(* PLC project Unnamed, Unknown Unnamed 1 *)
(* stored: creationDateTime 2024-01-09T16:45:07, modificationDateTime 2024-01-23T14:31:54 *)

FUNCTION_BLOCK Reals_Min
  VAR_INPUT
    u1 : REAL;
    u2 : REAL;
  END_VAR
  VAR_OUTPUT
    y : REAL;
  END_VAR

						y := min(u1, u2);
					
END_FUNCTION_BLOCK

FUNCTION_BLOCK Reals_MultiplyByParameter
  VAR_INPUT
    u : REAL;
    k : REAL;
  END_VAR
  VAR_OUTPUT
    y : REAL;
  END_VAR

						y := k * u;
					
END_FUNCTION_BLOCK

PROGRAM CustomPWithLimiter
  VAR_INPUT
    e : REAL;
    yMax : REAL;
  END_VAR
  VAR_OUTPUT
    y : REAL;
  END_VAR
  VAR
    gain : Reals_MultiplyByParameter;
    minValue : Reals_Min;
    k : REAL := 2.0;
  END_VAR

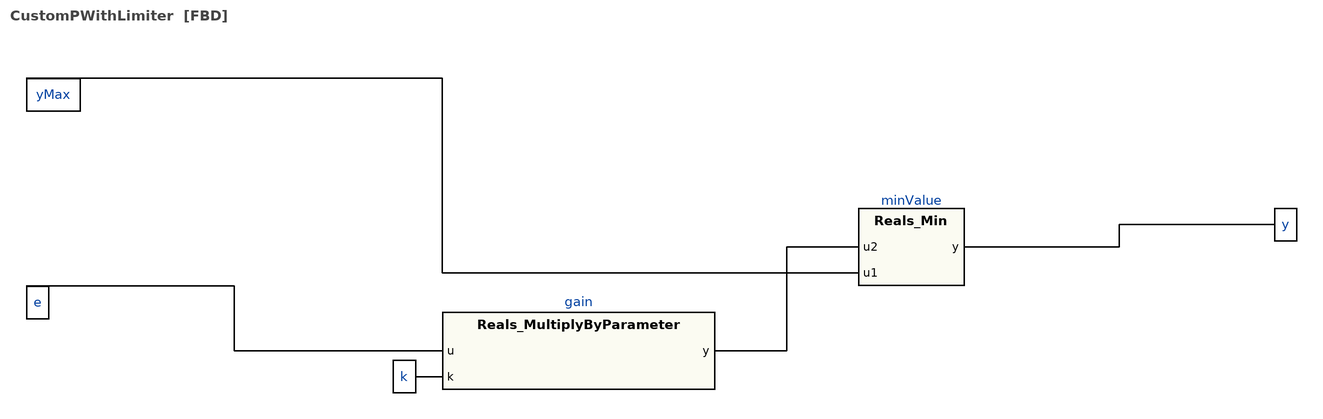
(* FBD diagram, written out as Structured Text *)
gain(u := e, k := k);
minValue(u2 := gain.y, u1 := yMax);
y := minValue.y;
END_PROGRAM

CONFIGURATION config
  RESOURCE resource1 ON PLC
    TASK task0(INTERVAL := T#20ms, PRIORITY := 0);
    PROGRAM instance0 WITH task0 : CustomPWithLimiter;
  END_RESOURCE
END_CONFIGURATION
